(* Logix 5000 project; controller L306 vendor 1 type 14 code 196 rev 32.12; software revision 32.02 *)

TASK MainTask (continuous, watchdog 500 ms) : MainProgram

MODULES
   Local : vendor 1 type 14 code 196 (5069 0, rev 32.12)
      VSD_AFE : vendor 1 type 143 code 8080 (Ethernet 192.168.2.150, rev 10.1, Output RPI 20 ms)
          : vendor 1 type 143 code 1697 (RhinoBP 10, rev 1.1)
          : vendor 1 type 143 code 4514 (RhinoBP 12, rev 1.1)
          : vendor 1 type 143 code 419 (RhinoBP 13, rev 1.1)
          : vendor 1 type 143 code 2468 (RhinoBP 14, rev 1.1)
      IO_Analog_Input : 5069-IF8 (5069 3, rev 2.1, StandardDataDriven RPI 100 ms)
      IO_Digital_In : 5069-IB16 (5069 1, rev 2.1, StandardDataDriven RPI 5 ms)
      IO_Digital_Out : vendor 1 type 7 code 1213 (5069 2, rev 3.1, StandardDataDriven RPI 5 ms)
END_MODULES

TYPE Dinagrama :   // Estructura para el dinagrama
STRUCT
   vPotencia : REAL[500];   // captura del vector de potencia
   vCarga : REAL[500];   // captura del vector de carga
   vPosicion : REAL[500];   // captura del vector posicion
   vProximetro : DINT[500];   // captura del vector del proximetro
   NumeroMuestras : INT;
   enabled : BOOL;
   captura : BOOL;   // Flag que indica la captura del sistema
   resetVector : BOOL;   // Flag para darle Reset al vector de posición y carga
   vEmptyREAL : REAL[500];
   vEmptyINT : DINT[500];
   tMuestreo : REAL;   // Tiempo de Muestreo de captura
END_STRUCT
END_TYPE

TYPE SWC :
STRUCT
   Dinagrama : Dinagrama;
   entradasDigitales : INT;
   salidasDigitales : INT;
   entradasAnalogas : REAL[4];
   salidasAnalogas : REAL[4];
   VSD : VSD;   // Comandos de Pantalla
END_STRUCT
END_TYPE

TYPE VSD :
STRUCT
   LogicCommand_Start : BOOL;
   LogicCommand_Stop : BOOL;
   LogicCommand_ClearFaults : BOOL;
   LogicCommand_Forward : BOOL;
   LogicCommand_Reverse : BOOL;
   Reference : REAL;
END_STRUCT
END_TYPE

VAR_GLOBAL   (* controller tags *)
   SWC : SWC := (Dinagrama.tMuestreo := 0.05, salidasDigitales := 1, VSD.Reference := 36.0);
END_VAR

PROGRAM MainProgram   (* main routine R000_MainRoutine *)

ROUTINE R000_MainRoutine   (* ladder *)
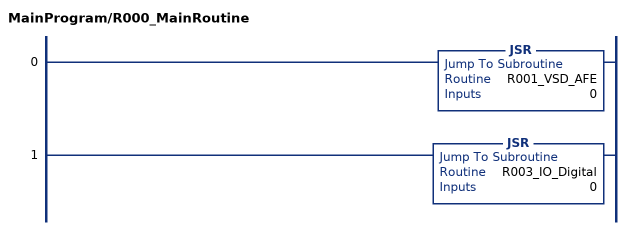
   0: JSR(R001_VSD_AFE,0);
   1: JSR(R003_IO_Digital,0);
END_ROUTINE

ROUTINE R001_VSD_AFE   (* ladder *)
// Comandos Basicos de Operación de VSD AFE
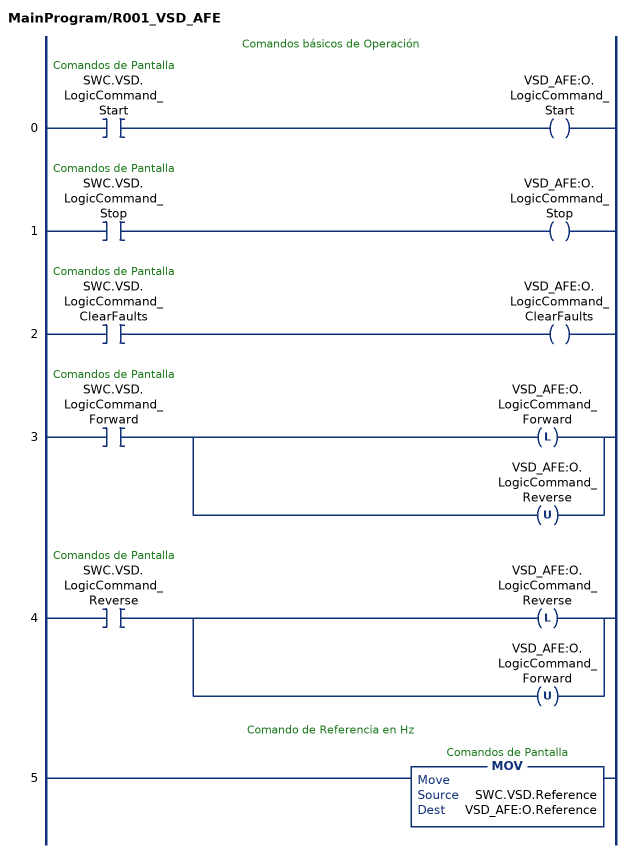
   // Comandos básicos de Operación
   0: XIC(SWC.VSD.LogicCommand_Start)OTE(VSD_AFE:O.LogicCommand_Start);
   1: XIC(SWC.VSD.LogicCommand_Stop)OTE(VSD_AFE:O.LogicCommand_Stop);
   2: XIC(SWC.VSD.LogicCommand_ClearFaults)OTE(VSD_AFE:O.LogicCommand_ClearFaults);
   3: XIC(SWC.VSD.LogicCommand_Forward)[OTL(VSD_AFE:O.LogicCommand_Forward) ,OTU(VSD_AFE:O.LogicCommand_Reverse) ];
   4: XIC(SWC.VSD.LogicCommand_Reverse)[OTL(VSD_AFE:O.LogicCommand_Reverse) ,OTU(VSD_AFE:O.LogicCommand_Forward) ];
   // Comando de Referencia en Hz
   5: MOV(SWC.VSD.Reference,VSD_AFE:O.Reference);
END_ROUTINE

ROUTINE R003_IO_Digital   (* ladder *)
// Entradas Digitales
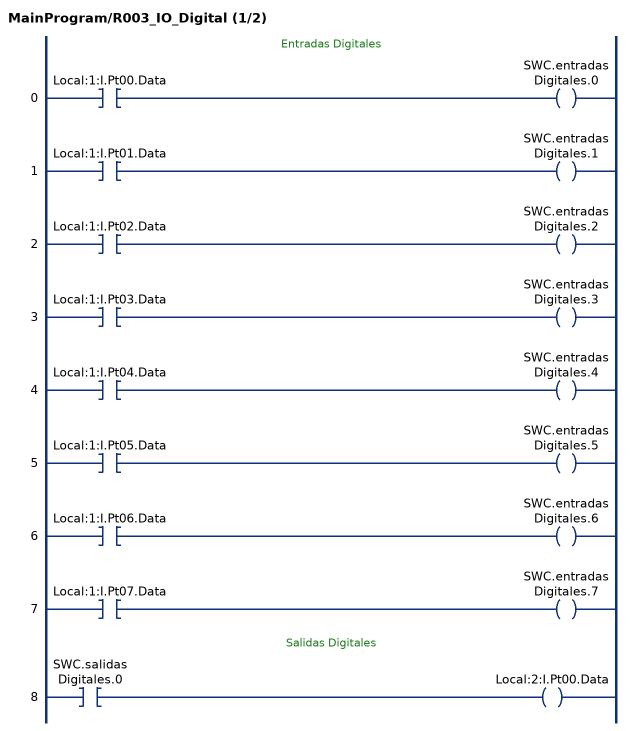
   // Entradas Digitales
   0: XIC(Local:1:I.Pt00.Data)OTE(SWC.entradasDigitales.0);
   1: XIC(Local:1:I.Pt01.Data)OTE(SWC.entradasDigitales.1);
   2: XIC(Local:1:I.Pt02.Data)OTE(SWC.entradasDigitales.2);
   3: XIC(Local:1:I.Pt03.Data)OTE(SWC.entradasDigitales.3);
   4: XIC(Local:1:I.Pt04.Data)OTE(SWC.entradasDigitales.4);
   5: XIC(Local:1:I.Pt05.Data)OTE(SWC.entradasDigitales.5);
   6: XIC(Local:1:I.Pt06.Data)OTE(SWC.entradasDigitales.6);
   7: XIC(Local:1:I.Pt07.Data)OTE(SWC.entradasDigitales.7);
   // Salidas Digitales
   8: XIC(SWC.salidasDigitales.0)OTE(Local:2:I.Pt00.Data);
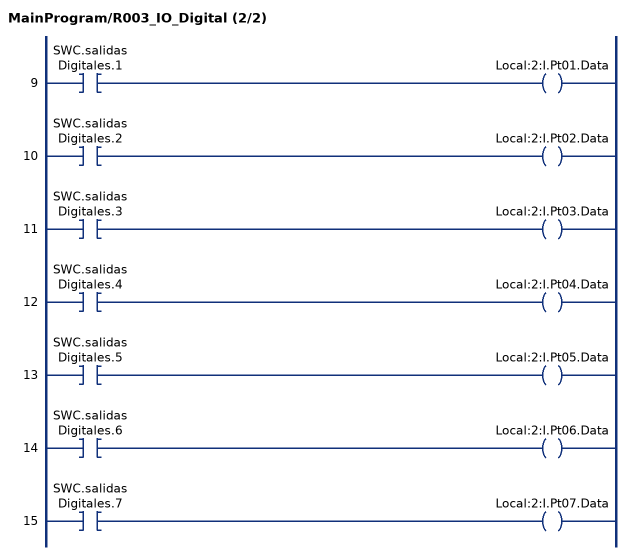
   9: XIC(SWC.salidasDigitales.1)OTE(Local:2:I.Pt01.Data);
   10: XIC(SWC.salidasDigitales.2)OTE(Local:2:I.Pt02.Data);
   11: XIC(SWC.salidasDigitales.3)OTE(Local:2:I.Pt03.Data);
   12: XIC(SWC.salidasDigitales.4)OTE(Local:2:I.Pt04.Data);
   13: XIC(SWC.salidasDigitales.5)OTE(Local:2:I.Pt05.Data);
   14: XIC(SWC.salidasDigitales.6)OTE(Local:2:I.Pt06.Data);
   15: XIC(SWC.salidasDigitales.7)OTE(Local:2:I.Pt07.Data);
END_ROUTINE
END_PROGRAM
